// TIA Portal V19 export
TYPE "LAF_typeXXXProcessValues"
// stored: Access Published
   STRUCT
      pieceCount : DInt;
   END_STRUCT;
END_TYPE
